SYSTEM Nutrunner
  (* Version 1.0, Author, 4DIAC-Consortium *)
  APPLICATION end2end
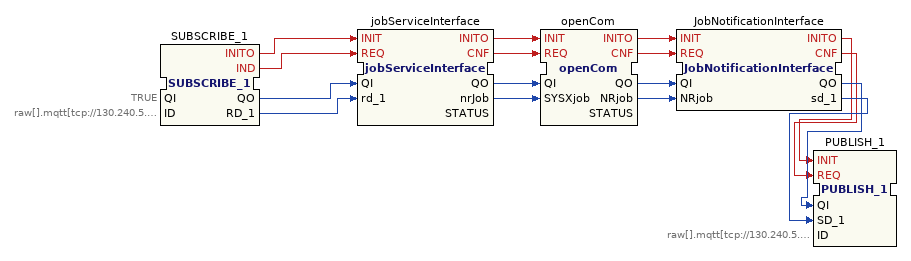
    FBS
      openCom : openCom;
      SUBSCRIBE_1 : SUBSCRIBE_1(QI := TRUE, ID := raw[].mqtt[tcp://130.240.5.130:1883,4diac,jobs]);
      PUBLISH_1 : PUBLISH_1(ID := raw[].mqtt[tcp://130.240.5.130:1883,4diac,jobs]);
      JobNotificationInterface : JobNotificationInterface;
      jobServiceInterface : jobServiceInterface;
    END_FBS
    EVENT_CONNECTIONS
      SUBSCRIBE_1.INITO TO jobServiceInterface.INIT;
      SUBSCRIBE_1.IND TO jobServiceInterface.REQ;
      jobServiceInterface.INITO TO openCom.INIT;
      jobServiceInterface.CNF TO openCom.REQ;
      openCom.INITO TO JobNotificationInterface.INIT;
      JobNotificationInterface.INITO TO PUBLISH_1.INIT;
      JobNotificationInterface.CNF TO PUBLISH_1.REQ;
      openCom.CNF TO JobNotificationInterface.REQ;
    END_CONNECTIONS
    DATA_CONNECTIONS
      SUBSCRIBE_1.QO TO jobServiceInterface.QI;
      SUBSCRIBE_1.RD_1 TO jobServiceInterface.rd_1;
      jobServiceInterface.nrJob TO openCom.SYSXjob;
      jobServiceInterface.QO TO openCom.QI;
      openCom.QO TO JobNotificationInterface.QI;
      openCom.NRjob TO JobNotificationInterface.NRjob;
      JobNotificationInterface.QO TO PUBLISH_1.QI;
      JobNotificationInterface.sd_1 TO PUBLISH_1.SD_1;
    END_CONNECTIONS
  END_APPLICATION
  DEVICE BeagleBoneBlack : BeagleBoneBlack(MGR_ID := "192.168.7.2:61499")
    {SET_ATTRIBUTE(Profile, HOLOBLOC)}
    RESOURCE EMB_RES : EMB_RES
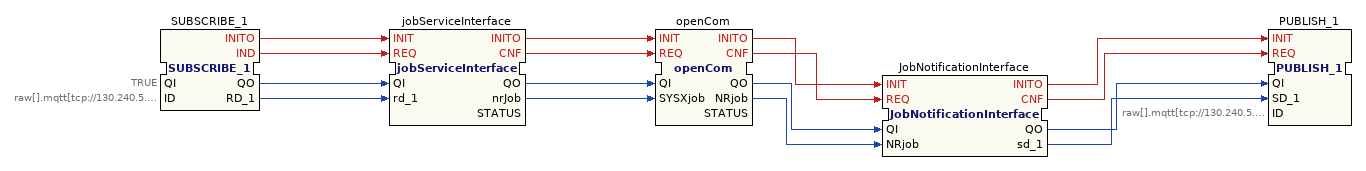
      FBS
        openCom : openCom;
        PUBLISH_1 : PUBLISH_1(ID := raw[].mqtt[tcp://130.240.5.130:1883,4diac,jobs]);
        SUBSCRIBE_1 : SUBSCRIBE_1(QI := TRUE, ID := raw[].mqtt[tcp://130.240.5.130:1883,4diac,jobs]);
        jobServiceInterface : jobServiceInterface;
        JobNotificationInterface : JobNotificationInterface;
      END_FBS
      EVENT_CONNECTIONS
        SUBSCRIBE_1.INITO TO jobServiceInterface.INIT;
        SUBSCRIBE_1.IND TO jobServiceInterface.REQ;
        jobServiceInterface.INITO TO openCom.INIT;
        jobServiceInterface.CNF TO openCom.REQ;
        openCom.INITO TO JobNotificationInterface.INIT;
        JobNotificationInterface.INITO TO PUBLISH_1.INIT;
        JobNotificationInterface.CNF TO PUBLISH_1.REQ;
        openCom.CNF TO JobNotificationInterface.REQ;
      END_CONNECTIONS
      DATA_CONNECTIONS
        SUBSCRIBE_1.QO TO jobServiceInterface.QI;
        SUBSCRIBE_1.RD_1 TO jobServiceInterface.rd_1;
        jobServiceInterface.nrJob TO openCom.SYSXjob;
        jobServiceInterface.QO TO openCom.QI;
        openCom.QO TO JobNotificationInterface.QI;
        openCom.NRjob TO JobNotificationInterface.NRjob;
        JobNotificationInterface.QO TO PUBLISH_1.QI;
        JobNotificationInterface.sd_1 TO PUBLISH_1.SD_1;
      END_CONNECTIONS
    END_RESOURCE
  END_DEVICE
  MAPPINGS
    end2end.openCom ON BeagleBoneBlack.EMB_RES.openCom;
    end2end.SUBSCRIBE_1 ON BeagleBoneBlack.EMB_RES.SUBSCRIBE_1;
    end2end.PUBLISH_1 ON BeagleBoneBlack.EMB_RES.PUBLISH_1;
    end2end.JobNotificationInterface ON BeagleBoneBlack.EMB_RES.JobNotificationInterface;
    end2end.jobServiceInterface ON BeagleBoneBlack.EMB_RES.jobServiceInterface;
  END_MAPPINGS
  SEGMENTS
    Ethernet : Ethernet;
  END_SEGMENTS
  LINKS
    BeagleBoneBlack => Ethernet;
  END_LINKS
END_SYSTEM
